Omron CX-Programmer project NewProject (CX-Programmer 9.61)

# PLC proyekTugas: CP1E NA

## Global symbols (name address type ; comment)
0.00 BOOL  ; start
0.01 BOOL  ; stop
0.02 BOOL  ; sensor 1
0.03 BOOL  ; Sensor Logam
0.04 BOOL  ; Non Logam
0.05 BOOL  ; Sensor output 1
0.06 BOOL  ; Sensor Output 2
0.07 BOOL  ; Hitung Reject
0.08 BOOL  ; Emergency
0.09 BOOL  ; start manual
0.10 BOOL  ; start and stop motor 1
0.11 BOOL  ; start and stop motor 2
0.12 BOOL  ; start and stop motor 3
0.13 BOOL  ; Sensor logam
0.14 BOOL  ; Sensor Non-Logam
100.00 BOOL  ; Konveyor 1 On
100.01 BOOL  ; Konveyor 2 On
100.02 BOOL  ; Konveyor 3 On
100.03 BOOL  ; robot 1
100.04 BOOL  ; robot 2
100.05 BOOL  ; robot 1
10.00 BOOL  ; system otomatis
20.00 BOOL  ; Kunci jika lama menunggu
50.00 BOOL  ; system manual
T000 BOOL  ; waktu lama konveyor berkerja
T003 BOOL  ; waktu robot1
T004 BOOL  ; waktu robot 2
T005 BOOL  ; Robot 2

## Program NewProgram1 (cyclic task 0)
Local symbols
d BOOL

### Section Section1

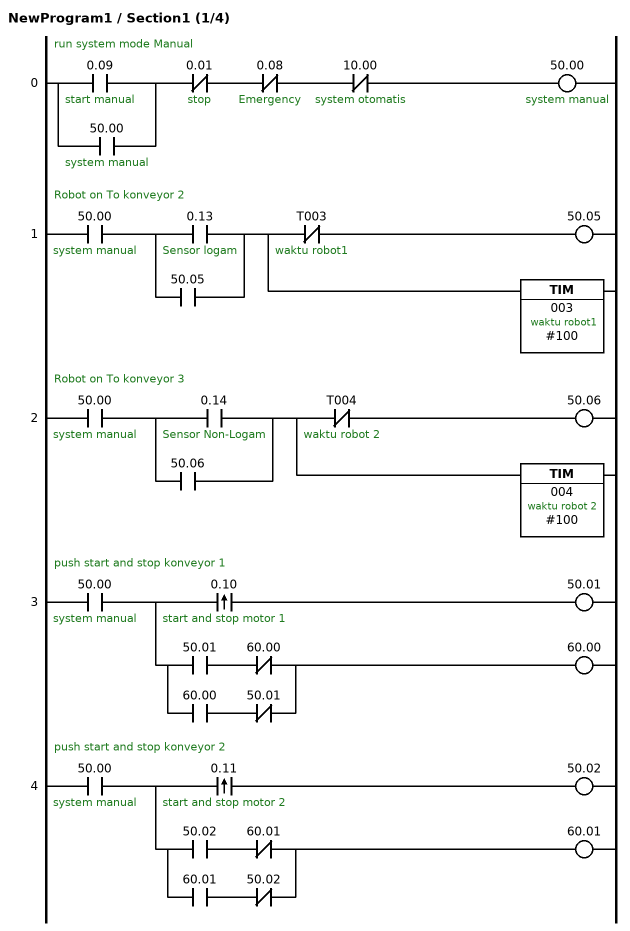
; rung 0: run system mode Manual
LD 0.09  ; start manual
OR 50.00  ; system manual
ANDNOT 0.01  ; stop
ANDNOT 0.08  ; Emergency
ANDNOT 10.00  ; system otomatis
OUT 50.00  ; system manual
; rung 1: Robot on To konveyor 2
LD 50.00  ; system manual
LD 0.13  ; Sensor logam
OR 50.05
ANDLD
OUT TR0
ANDNOT T003  ; waktu robot1
OUT 50.05
LD TR0
TIM 003 #100  ; waktu robot1
; rung 2: Robot on To konveyor 3
LD 50.00  ; system manual
LD 0.14  ; Sensor Non-Logam
OR 50.06
ANDLD
OUT TR0
ANDNOT T004  ; waktu robot 2
OUT 50.06
LD TR0
TIM 004 #100  ; waktu robot 2
; rung 3: push start and stop konveyor 1
LD 50.00  ; system manual
OUT TR0
@AND 0.10  ; start and stop motor 1
OUT 50.01
LD TR0
LD 50.01
ANDNOT 60.00
LD 60.00
ANDNOT 50.01
ORLD
ANDLD
OUT 60.00
; rung 4: push start and stop konveyor 2
LD 50.00  ; system manual
OUT TR0
@AND 0.11  ; start and stop motor 2
OUT 50.02
LD TR0
LD 50.02
ANDNOT 60.01
LD 60.01
ANDNOT 50.02
ORLD
ANDLD
OUT 60.01

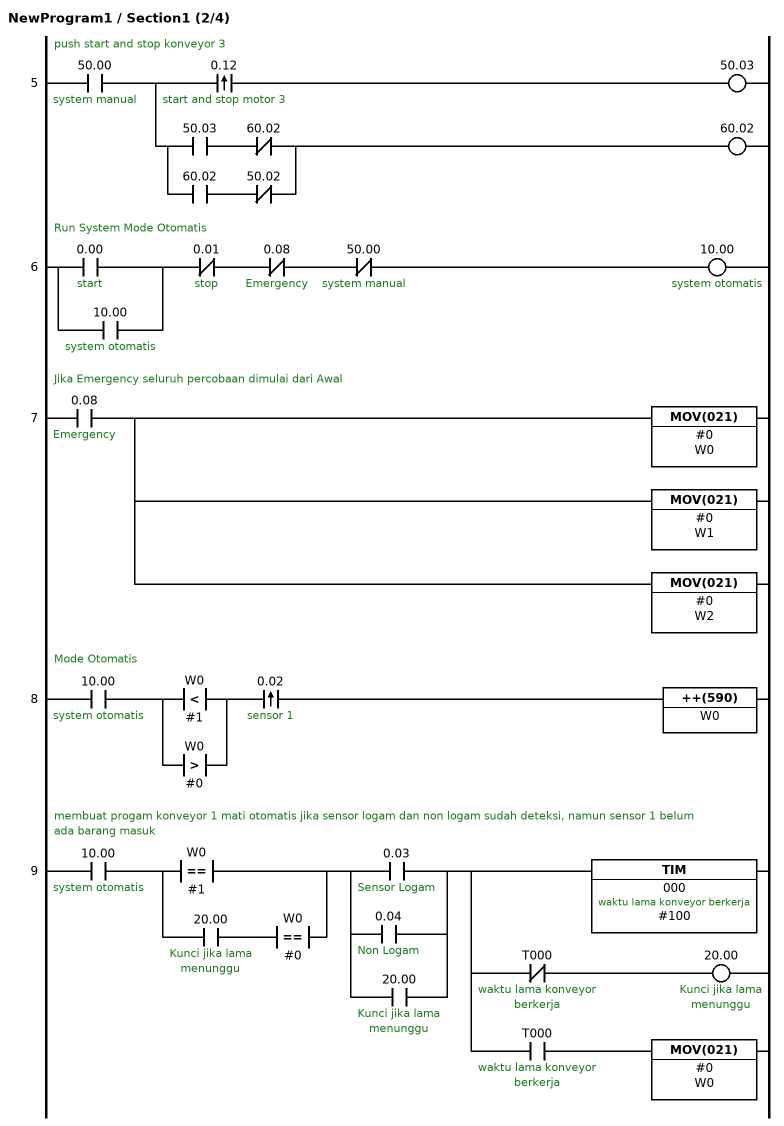
; rung 5: push start and stop konveyor 3
LD 50.00  ; system manual
OUT TR0
@AND 0.12  ; start and stop motor 3
OUT 50.03
LD TR0
LD 50.03
ANDNOT 60.02
LD 60.02
ANDNOT 50.02
ORLD
ANDLD
OUT 60.02
; rung 6: Run System Mode Otomatis
LD 0.00  ; start
OR 10.00  ; system otomatis
ANDNOT 0.01  ; stop
ANDNOT 0.08  ; Emergency
ANDNOT 50.00  ; system manual
OUT 10.00  ; system otomatis
; rung 7: Jika Emergency seluruh percobaan dimulai dari Awal
LD 0.08  ; Emergency
MOV(021) #0 W0
MOV(021) #0 W1
MOV(021) #0 W2
; rung 8: Mode Otomatis
LD 10.00  ; system otomatis
LD<(310) W0 #1
OR>(320) W0 #0
ANDLD
@AND 0.02  ; sensor 1
++(590) W0
; rung 9: membuat progam konveyor 1 mati otomatis jika sensor logam dan non logam sudah deteksi, namun sensor 1 belum ada barang masuk
LD 10.00  ; system otomatis
LD=(300) W0 #1
LD 20.00  ; Kunci jika lama menunggu
AND=(300) W0 #0
ORLD
ANDLD
LD 0.03  ; Sensor Logam
OR 0.04  ; Non Logam
OR 20.00  ; Kunci jika lama menunggu
ANDLD
OUT TR0
TIM 000 #100  ; waktu lama konveyor berkerja
ANDNOT T000  ; waktu lama konveyor berkerja
OUT 20.00  ; Kunci jika lama menunggu
LD TR0
AND T000  ; waktu lama konveyor berkerja
MOV(021) #0 W0

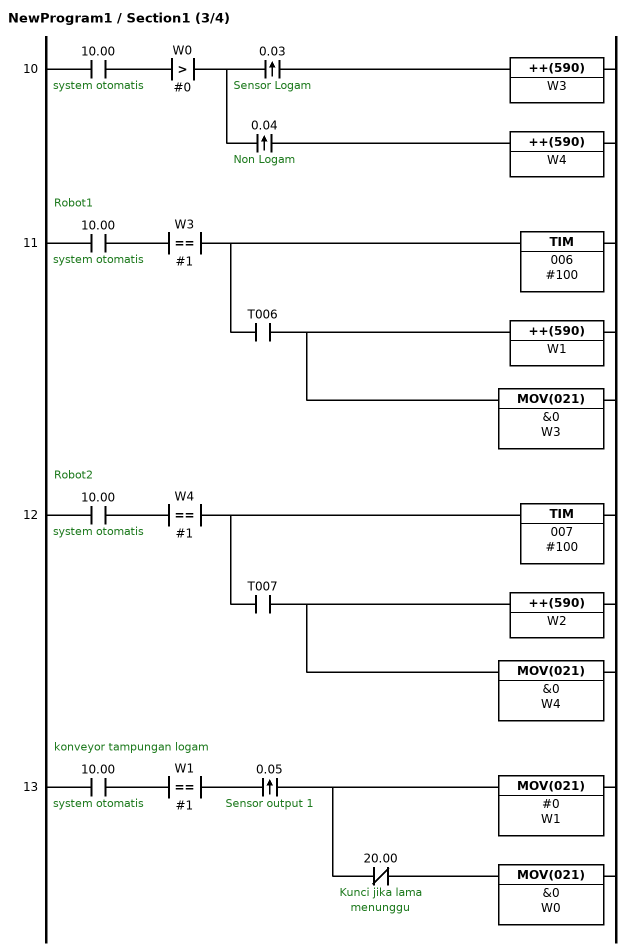
; rung 10
LD 10.00  ; system otomatis
AND>(320) W0 #0
OUT TR0
@AND 0.03  ; Sensor Logam
++(590) W3
LD TR0
@AND 0.04  ; Non Logam
++(590) W4
; rung 11: Robot1
LD 10.00  ; system otomatis
AND=(300) W3 #1
TIM 006 #100
AND T006
++(590) W1
MOV(021) &0 W3
; rung 12: Robot2
LD 10.00  ; system otomatis
AND=(300) W4 #1
TIM 007 #100
AND T007
++(590) W2
MOV(021) &0 W4
; rung 13: konveyor tampungan logam
LD 10.00  ; system otomatis
AND=(300) W1 #1
@AND 0.05  ; Sensor output 1
MOV(021) #0 W1
ANDNOT 20.00  ; Kunci jika lama menunggu
MOV(021) &0 W0

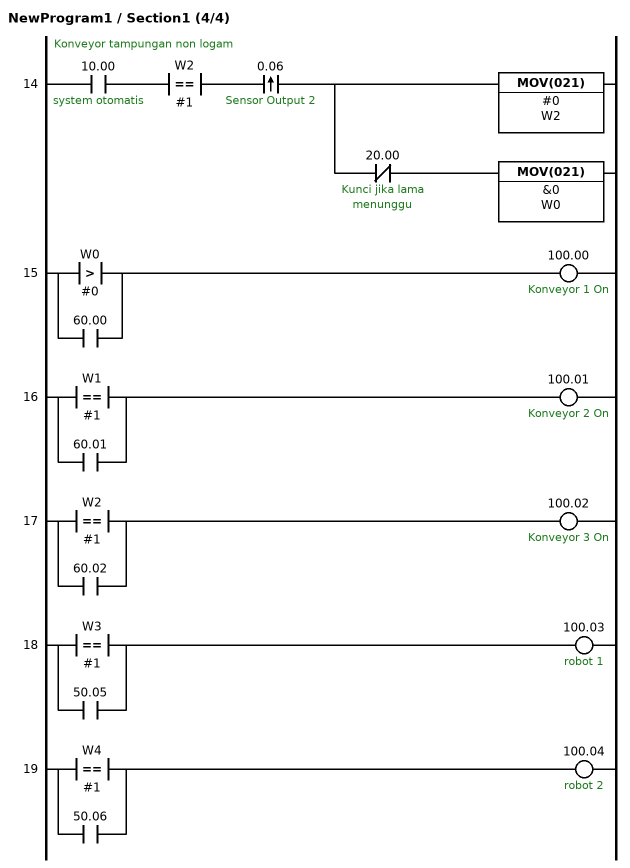
; rung 14: Konveyor tampungan non logam
LD 10.00  ; system otomatis
AND=(300) W2 #1
@AND 0.06  ; Sensor Output 2
MOV(021) #0 W2
ANDNOT 20.00  ; Kunci jika lama menunggu
MOV(021) &0 W0
; rung 15
LD>(320) W0 #0
OR 60.00
OUT 100.00  ; Konveyor 1 On
; rung 16
LD=(300) W1 #1
OR 60.01
OUT 100.01  ; Konveyor 2 On
; rung 17
LD=(300) W2 #1
OR 60.02
OUT 100.02  ; Konveyor 3 On
; rung 18
LD=(300) W3 #1
OR 50.05
OUT 100.03  ; robot 1
; rung 19
LD=(300) W4 #1
OR 50.06
OUT 100.04  ; robot 2

### Section END
; rung 0
END(001)